Universal Robots PolyScope program: Lower_Z.urp

Program Lower_Z (installation=default directory=/programs/usbdisk createdIn=3.15.4.106291 lastSavedIn=3.15.4.106291 robotSerialNumber=2019300133)
Calibrated DH parameters: a=[-0.000006, -0.606471, -0.570201, -0.000053, 0.000006, 0]; d=[0.128096, 15.114888, -22.674746, 7.723348, 0.115665, 0.092162]; alpha=[1.570605, -0.005579, -0.004649, 1.571049, -1.571015, 0]; deltaTheta=[-0.00004, -0.169247, 0.199673, -0.061563, -0.000077, -0.000043]
Robot Program (runOnlyOnce=false)
  Script: current_pose = get_actual_tcp_pose()
  URCap Conveyor Tracking (Conveyor Tracking, Universal Robots)
    Script: new_pose = p[current_pose[0], current_pose[1], current_pose[2] + 0.1, current_pose[3] , current_pose[4], current_pose[5]]
    Script: movej(new_pose , a = 0.1, v =0.1)
